TYPE E_SignalMode :
(

	SignalMode_Off,
    SignalMode_Static,
    SignalMode_Rectangle,
    SignalMode_Sinus,
    SignalMode_Triangle
   
);
END_TYPE

(* stored: Version 1.1.0.1, ProductVersion 3.1.4026.12
   DUT E_SignalMode: Id {54c7c7ec-8552-4782-8ae3-168155635a5a} *)
